FUNCTION F_SineFunction_secondary : LREAL
VAR_INPUT
	fTime 				: LREAL;
END_VAR
VAR_OUTPUT
	fSineSignal 		: LREAL;
END_VAR
VAR
	u					: LREAL;
	ft_ENV				: LREAL := 3.0;
	y					: LREAL;
	
END_VAR

(*u := fTime/ft_ENV;

IF u > 1.0 THEN
	u := 1.0;
END_IF

y := (3.0*u*u) - (2.0*u*u*u);*)

fSineSignal := G_Engineer_HMI.fAmp * SIN(2.0 * PI * G_Engineer_HMI.fFreq * fTime) + G_Engineer_HMI.fSinemidpoint; //y gange i starten om soft start skal på

END_FUNCTION

(* stored: Version 1.1.0.1
   POU F_SineFunction_secondary: Id {649bd89c-704c-46cd-9a20-ba5de6666f89}, SpecialFunc None *)
